FUNCTION_BLOCK FB_SensorBinary_Test EXTENDS TcUnit.FB_TestSuite
VAR
	fbSensorBinary : FB_SensorBinary;
	nExpected : BYTE;
	nResult : BYTE;
	bExpected : BOOL;
	bResult : BOOL;
END_VAR

TEST('Get bValue FALSE');
fbSensorBinary.SetStatus(0);
fbSensorBinary();
bExpected := FALSE;
bResult := fbSensorBinary.bValue;

AssertEquals(Expected := bExpected,
             Actual := bResult,
             Message := 'Value is not correct');	
TEST_FINISHED();

TEST('Get bValue TRUE');	
fbSensorBinary.SetStatus(1);
fbSensorBinary();
bExpected := 1;
bResult := fbSensorBinary.bValue;
AssertEquals(Expected := bExpected,
             Actual := bResult,
             Message := 'Control value is not correct');	 
TEST_FINISHED();

END_FUNCTION_BLOCK

(* stored: Version 1.1.0.1, ProductVersion 3.1.4024.12
   POU FB_SensorBinary_Test: Id {80045a0d-866a-0cac-3ab1-dd3a70d21b12}, SpecialFunc None *)
